// TIA Portal V17 export
// export: Created 2023-12-22T15:08:07.8686869Z, ExportSetting WithDefaults, DisplayName Totally Integrated Automation Portal, DisplayVersion V17, DisplayName TIA Portal Openness, DisplayVersion V17, DisplayName TIA Portal Version Control Interface, DisplayVersion V17, DisplayName STEP 7 Professional, DisplayVersion V17, DisplayName STEP 7 Safety, DisplayVersion V17, DisplayName WinCC Advanced, DisplayVersion V17
FUNCTION_BLOCK "Time_M"   // FB92, LAD
{ S7_Optimized_Access := 'FALSE' }
VERSION : 0.1
// stored: AutoNumber false, IsIECCheckEnabled false, SetENOAutomatically false, UDAEnableTagReadback false
   VAR DB_SPECIFIC
      SP_M { S7_SetPoint := 'True'} : Int;
      SP_S { S7_SetPoint := 'True'} : Int := 30;
      Now_M : Int;
      Now_S : Int;
      Rev_M : Int;
      Rev_S : Int;
      Progress : Real;
      Start : Bool;
      "Exit" : Bool;
      Pause : Bool;
      Reset : Bool;
   END_VAR
   VAR_TEMP
      Full_SP_S : Int;
      Full_Now_S : Int;
      Full_Delta_S : Int;
   END_VAR
   VAR_TEMP   // added for the SCL form of the ladder/FBD networks
      _w1 : Bool;
   END_VAR
BEGIN

REGION Network 1: Подсчёт времени
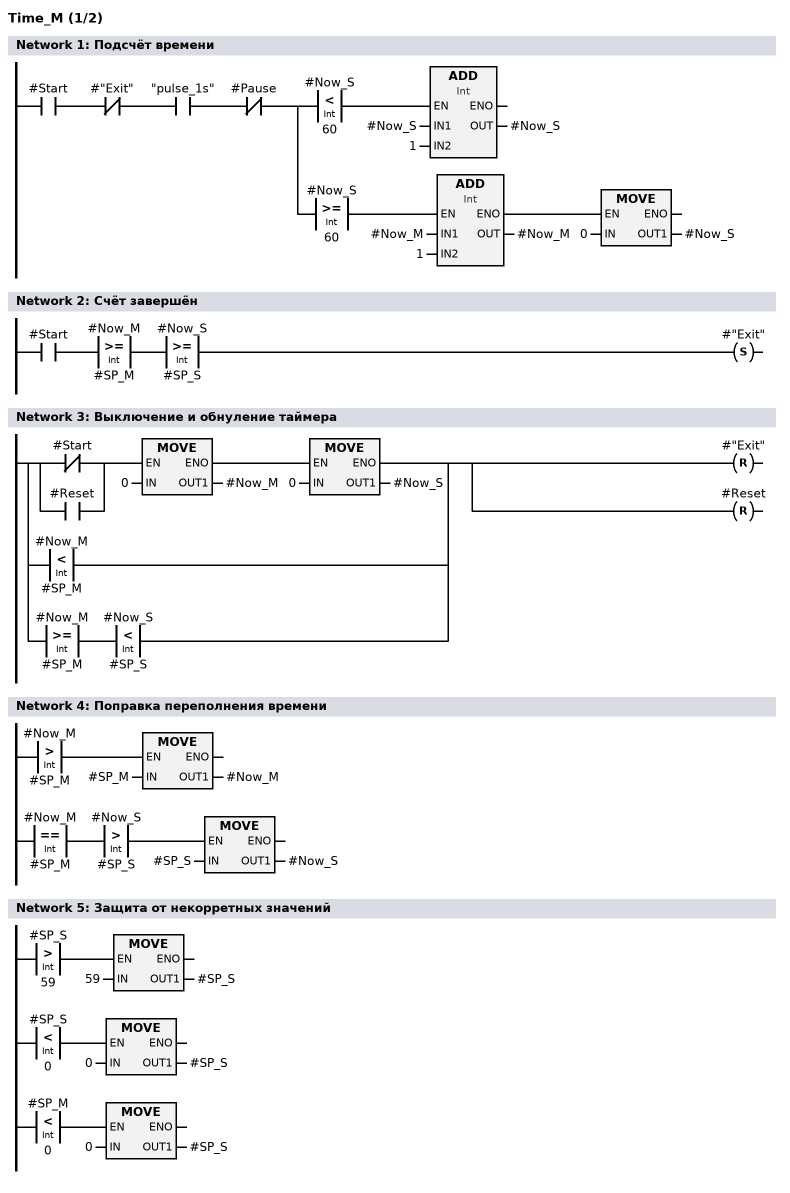
   RUNG wire#powerrail
      Contact( #Start )
      I_Contact( #"Exit" )
      Contact( "pulse_1s" )
      I_Contact( #Pause )
      wire#w1
      { S7_Templates := "SrcType := Int" } LT_Contact(in1 := #Now_S, in2 := 60)
      { S7_Templates := "SrcType := Int"; S7_GenerateENO := "TRUE" } Add(in1 := #Now_S, in2 := 1, out => #Now_S)
   END_RUNG
   RUNG wire#w1
      { S7_Templates := "SrcType := Int" } GE_Contact(in1 := #Now_S, in2 := 60)
      { S7_Templates := "SrcType := Int"; S7_GenerateENO := "TRUE" } Add(in1 := #Now_M, in2 := 1, out => #Now_M)
      { S7_GenerateENO := "TRUE" } Move(in := 0, out1 => #Now_S)
   END_RUNG
   // the same network as SCL:
   // ENO of a box is taken as its EN; it also drops when the box reports an error
   #_w1 := #Start AND NOT #"Exit" AND "pulse_1s" AND NOT #Pause;
   IF #_w1 AND (#Now_S < 60) THEN #Now_S := #Now_S + 1; END_IF;
   IF #_w1 AND (#Now_S >= 60) THEN
       #Now_M := #Now_M + 1;
       #Now_S := 0;
   END_IF;
END_REGION

REGION Network 2: Счёт завершён
   RUNG wire#powerrail
      Contact( #Start )
      { S7_Templates := "SrcType := Int" } GE_Contact(in1 := #Now_M, in2 := #SP_M)
      { S7_Templates := "SrcType := Int" } GE_Contact(in1 := #Now_S, in2 := #SP_S)
      S_Coil( #"Exit" )
   END_RUNG
   // the same network as SCL:
   IF #Start AND (#Now_M >= #SP_M) AND (#Now_S >= #SP_S) THEN #"Exit" := TRUE; END_IF;
END_REGION

REGION Network 3: Выключение и обнуление таймера
   RUNG wire#powerrail
      I_Contact( #Start )
      wire#w1
      { S7_GenerateENO := "TRUE" } Move(in := 0, out1 => #Now_M)
      { S7_GenerateENO := "TRUE" } Move(in := 0, out1 => #Now_S)
      wire#w2
      R_Coil( #"Exit" )
   END_RUNG
   RUNG wire#powerrail
      Contact( #Reset )
   END_RUNG wire#w1
   RUNG wire#powerrail
      { S7_Templates := "SrcType := Int" } LT_Contact(in1 := #Now_M, in2 := #SP_M)
   END_RUNG wire#w2
   RUNG wire#powerrail
      { S7_Templates := "SrcType := Int" } GE_Contact(in1 := #Now_M, in2 := #SP_M)
      { S7_Templates := "SrcType := Int" } LT_Contact(in1 := #Now_S, in2 := #SP_S)
   END_RUNG wire#w2
   RUNG wire#w2
      R_Coil( #Reset )
   END_RUNG
   // the same network as SCL:
   // ENO of a box is taken as its EN; it also drops when the box reports an error
   #_w1 := NOT #Start OR #Reset;
   IF #_w1 THEN
       #Now_M := 0;
       #Now_S := 0;
   END_IF;
   IF #_w1 OR (#Now_M < #SP_M) OR ((#Now_M >= #SP_M) AND (#Now_S < #SP_S)) THEN
       #"Exit" := FALSE;
       #Reset := FALSE;
   END_IF;
END_REGION

REGION Network 4: Поправка переполнения времени
   RUNG wire#powerrail
      { S7_Templates := "SrcType := Int" } GT_Contact(in1 := #Now_M, in2 := #SP_M)
      { S7_GenerateENO := "TRUE" } Move(in := #SP_M, out1 => #Now_M)
   END_RUNG
   RUNG wire#powerrail
      { S7_Templates := "SrcType := Int" } EQ_Contact(in1 := #Now_M, in2 := #SP_M)
      { S7_Templates := "SrcType := Int" } GT_Contact(in1 := #Now_S, in2 := #SP_S)
      { S7_GenerateENO := "TRUE" } Move(in := #SP_S, out1 => #Now_S)
   END_RUNG
   // the same network as SCL:
   IF #Now_M > #SP_M THEN #Now_M := #SP_M; END_IF;
   IF (#Now_M = #SP_M) AND (#Now_S > #SP_S) THEN #Now_S := #SP_S; END_IF;
END_REGION

REGION Network 5: Защита от некорретных значений
   RUNG wire#powerrail
      { S7_Templates := "SrcType := Int" } GT_Contact(in1 := #SP_S, in2 := 59)
      { S7_GenerateENO := "TRUE" } Move(in := 59, out1 => #SP_S)
   END_RUNG
   RUNG wire#powerrail
      { S7_Templates := "SrcType := Int" } LT_Contact(in1 := #SP_S, in2 := 0)
      { S7_GenerateENO := "TRUE" } Move(in := 0, out1 => #SP_S)
   END_RUNG
   RUNG wire#powerrail
      { S7_Templates := "SrcType := Int" } LT_Contact(in1 := #SP_M, in2 := 0)
      { S7_GenerateENO := "TRUE" } Move(in := 0, out1 => #SP_S)
   END_RUNG
   // the same network as SCL:
   IF #SP_S > 59 THEN #SP_S := 59; END_IF;
   IF #SP_S < 0 THEN #SP_S := 0; END_IF;
   IF #SP_M < 0 THEN #SP_S := 0; END_IF;
END_REGION

REGION Network 6: Обратный отсчёт
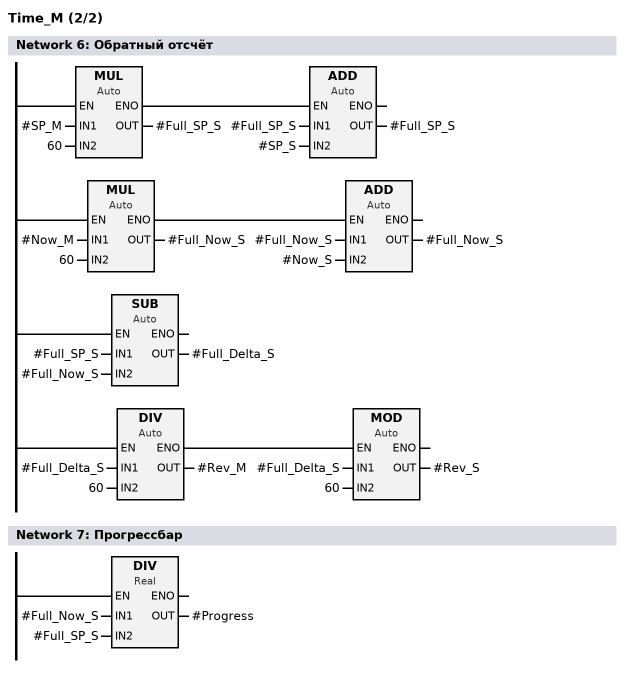
   RUNG wire#powerrail
      Mul(in1 := #SP_M, in2 := 60, out => #Full_SP_S)
      Add(in1 := #Full_SP_S, in2 := #SP_S, out => #Full_SP_S)
   END_RUNG
   RUNG wire#powerrail
      Mul(in1 := #Now_M, in2 := 60, out => #Full_Now_S)
      Add(in1 := #Full_Now_S, in2 := #Now_S, out => #Full_Now_S)
   END_RUNG
   RUNG wire#powerrail
      Sub(in1 := #Full_SP_S, in2 := #Full_Now_S, out => #Full_Delta_S)
   END_RUNG
   RUNG wire#powerrail
      Div(in1 := #Full_Delta_S, in2 := 60, out => #Rev_M)
      Mod(in1 := #Full_Delta_S, in2 := 60, out => #Rev_S)
   END_RUNG
   // the same network as SCL:
   #Full_SP_S := #SP_M * 60;
   #Full_SP_S := #Full_SP_S + #SP_S;
   #Full_Now_S := #Now_M * 60;
   #Full_Now_S := #Full_Now_S + #Now_S;
   #Full_Delta_S := #Full_SP_S - #Full_Now_S;
   #Rev_M := #Full_Delta_S / 60;
   #Rev_S := #Full_Delta_S MOD 60;
END_REGION

REGION Network 7: Прогрессбар
   RUNG wire#powerrail
      { S7_Templates := "SrcType := Real" } Div(in1 := #Full_Now_S, in2 := #Full_SP_S, out => #Progress)
   END_RUNG
   // the same network as SCL:
   #Progress := #Full_Now_S / #Full_SP_S;
END_REGION
END_FUNCTION_BLOCK
